// TIA Portal V16 export
// export: Created 2023-03-29T11:03:19.5147514Z, ExportSetting WithDefaults, DisplayName Totally Integrated Automation Portal, DisplayVersion V16 Update 6, DisplayName TIA Portal Version Control Interface, DisplayVersion V16 Update 2, DisplayName TIA Portal Openness, DisplayVersion V16 Update 6, DisplayName STEP 7 Professional, DisplayVersion V16 Update 6, DisplayName STEP 7 Safety, DisplayVersion V16, DisplayName WinCC Advanced, DisplayVersion V16 Update 6
DATA_BLOCK "DB31_HMI_AreaPointer"   // DB31
{ S7_Optimized_Access := 'FALSE' }
VERSION : 0.1
// stored: AutoNumber false, DBAccessibleFromOPCUA true, IsOnlyStoredInLoadMemory false, IsWriteProtectedInAS false
   VAR
      Coordination : Word;
      DateTime : DTL;
      JobMailbox : Array[0..3] of Word;
      DataRecord : Array[0..4] of Word;
      ProjectID : Word;
      ScreenNumber : Array[0..4] of Word;
      DateTimePLC : Struct
         DateTime : DTL;
         Reserve_01 : Word;
         Reserve_02 : Word;
      END_STRUCT;
      getPLCMode : Int;
      retValueTime : Word;
      cpuSatus : Bool;   // bit satus CPU (0-RUN, 1-RESATR)
   END_VAR
BEGIN
END_DATA_BLOCK
